FUNCTION_BLOCK DeviationMonitor
VAR_INPUT
	EN: BOOL := TRUE;
	Value: LREAL;
	TargetValue: LREAL := 100;
	DiffAllowed: LREAL := 5;
	Mode: DeviationMonitorMode := DeviationMonitorMode.Diff;
	Hysteresis: LREAL := 2;
	OnDelay: LTIME := LTIME#10S;
	OffDelay: LTIME := LTIME#5S;
END_VAR
VAR_OUTPUT
	ENO: BOOL;
	Error: BOOL;
END_VAR
VAR
	TempError: BOOL;
	Hyst: Hysteresis;
	UseValue: LREAL;
	UseTargetValue: LREAL;
	OnTON: TON;
	OffTOF: TOF;
END_VAR

UseValue  := Value;
UseTargetValue := TargetValue;
IF Mode = DeviationMonitorMode.Diff THEN
	UseValue := ABS(UseValue - TargetValue);	
	UseTargetValue := DiffAllowed;
END_IF
Hyst(Value := UseValue, LimitValue := UseTargetValue, Offset := Hysteresis);
IF EN and (Main.GreenMaster.GetParameters().System.Operation.State = SystemStates.Run) THEN
	IF (Mode = DeviationMonitorMode.Above) OR (Mode = DeviationMonitorMode.Diff) THEN
		TempError := Hyst.Above;
	ELSIF Mode = DeviationMonitorMode.Below THEN
		TempError := Hyst.Below;	
	END_IF
	IF Main.GreenMaster.GetParameters().System.Operation.State <> SystemStates.Run THEN
		TempError := False;
	END_IF
	OnTON(IN := TempError, PT := TO_TIME(OnDelay));
	OffTOF(IN := NOT TempError, PT := TO_TIME(OnDelay));
	IF OnTON.Q THEN
		Error := TRUE;
	END_IF
	IF OffTOF.Q THEN
		Error := FALSE;
	END_IF
ELSE
	Error := FALSE;
END_IF
ENO := EN;

END_FUNCTION_BLOCK

(* stored: Version 1.1.0.1, ProductVersion 3.1.4024.6
   POU DeviationMonitor: Id {dcb4d293-8c24-4f80-8a3f-089ab8e38d9c}, SpecialFunc None *)
